FUNCTION_BLOCK RT_E_CYCLE (* Delayed propagation of an event-Cancellable *)
  (* Description: Copyright (c) 2008 ACIN This program and the accompanying materials are made available under the terms of the Eclipse Public License 2.0 which is available at https://www.eclipse.org/legal/epl-2.0/ SPDX-License-Identifier: EPL-2.0 *)
  (* Version 3.0, 2025-04-14, Patrick Aigner, changed package *)
  (* Version 1.0, 2008-07-10, Alois Zoitl, ACIN *)
  PACKAGE eclipse4diac::rtevents;
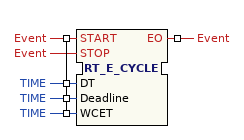
  EVENT_INPUT
    START WITH DT, Deadline, WCET; (* Begin Delay *)
    STOP; (* Cancel Delay *)
  END_EVENT
  EVENT_OUTPUT
    EO WITH QO; (* Delayed Event *)
  END_EVENT
  VAR_INPUT
    DT : TIME; (* Delay Time *)
    Deadline : TIME;
    WCET : TIME;
  END_VAR
END_FUNCTION_BLOCK
